FUNCTION_BLOCK FB_DryingPhase

VAR_INPUT
END_VAR

VAR_OUTPUT
	bDryingDone : BOOL;
END_VAR

VAR
END_VAR

//bDryingDone := (* Verdadeiro quando a etapa de secagem for concluída;

END_FUNCTION_BLOCK

(* stored: Version 1.1.0.1, ProductVersion 3.1.4024.13
   POU FB_DryingPhase: Id {3fed5c2e-00c0-41f9-b86a-23cb950cee48}, SpecialFunc None *)
